// TIA Portal V20 export
TYPE "typeNormalInterlockStatus"
// stored: Access Published, IsFailsafeCompliant true, Namespace Safety
   STRUCT
      BA10 : "Safety.s_zc_NormalInterlocks";
      BA15 : "Safety.s_zc_NormalInterlocks";
      BA40 : "Safety.s_zc_NormalInterlocks";
      BA60 : "Safety.s_zc_NormalInterlocks";
   END_STRUCT;
END_TYPE
